(* Schneider Machine Expert - Basic project resolucao, file version 2.7.0.0 *)
(* ProjectInformations: Name=Novo projeto *)

HARDWARE
  Cpu 0: TM221CE24R
  EthernetConfiguration: NetworkName=M221, IpAllocationMode=FixedAddress, IpAddress=0.0.0.0, SubnetMask=0.0.0.0
  SerialLineConfiguration: Baud=Baud19200, Parity=ParityEven, DataBits=DataBits8, StopBits=StopBits1, PhysicalMedium=PhysicalMediumRs485, TransmissionMode=TransmissionModeModbusRtu, SlaveId=1, Addressing=SlaveAddressing
  MastTask: UsePeriodScanMode=false, PeriodScan=100
  FastTask: Period=255
  CpuBehavior: StartingMode=StartAsPreviousState, AutoSaveRamOnEeprom=true, WatchdogPeriod=250

SYMBOLS  (address, symbol, comment, settings)
  %M0       SIG_IN_SEN_A
  %M1       SIG_IN_BOT_A
  %M10      SIG_OUT_EST_A_LIGA
  %M11      SIG_OUT_EST_A_DESL
  %TM0        [Preset=5, Base=OneSecond]
  %I0.0     IN_SEN_A
  %I0.1     IN_BOT_A
  %Q0.1     OUT_EST_A

POU Entradas
  (* SectionNumber=1 *)

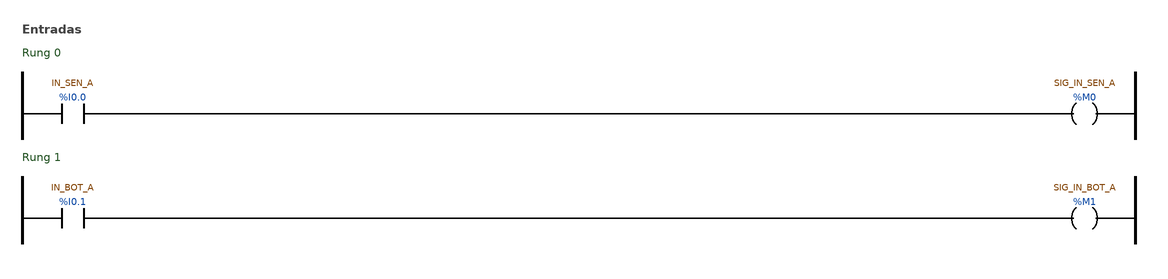

// Rung 0
  LD %I0.0                (* IN_SEN_A *)
  ST %M0                  (* SIG_IN_SEN_A *)
  // as ST:
  //   SIG_IN_SEN_A := IN_SEN_A;

// Rung 1
  LD %I0.1                (* IN_BOT_A *)
  ST %M1                  (* SIG_IN_BOT_A *)
  // as ST:
  //   SIG_IN_BOT_A := IN_BOT_A;

POU Lógicas
  (* SectionNumber=2 *)

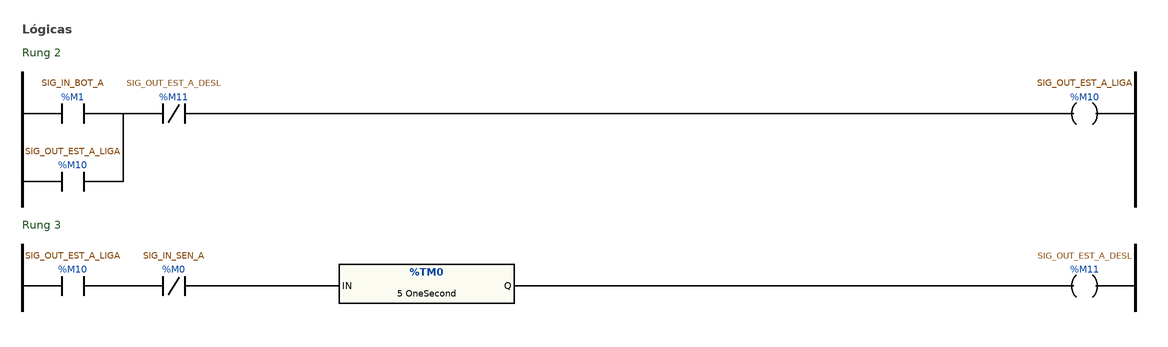

// Rung 2
  LD %M1                  (* SIG_IN_BOT_A *)
  OR %M10                 (* SIG_OUT_EST_A_LIGA *)
  ANDN %M11               (* SIG_OUT_EST_A_DESL *)
  ST %M10                 (* SIG_OUT_EST_A_LIGA *)
  // as ST:
  //   SIG_OUT_EST_A_LIGA := (SIG_IN_BOT_A OR SIG_OUT_EST_A_LIGA) AND NOT SIG_OUT_EST_A_DESL;

// Rung 3
  BLK %TM0
  LD %M10                 (* SIG_OUT_EST_A_LIGA *)
  ANDN %M0                (* SIG_IN_SEN_A *)
  IN
  OUT_BLK
  LD Q
  ST %M11                 (* SIG_OUT_EST_A_DESL *)
  END_BLK
  // as ST:
  //   %TM0(IN := SIG_OUT_EST_A_LIGA AND NOT SIG_IN_SEN_A);
  //   SIG_OUT_EST_A_DESL := %TM0.Q;

POU Saídas
  (* SectionNumber=3 *)

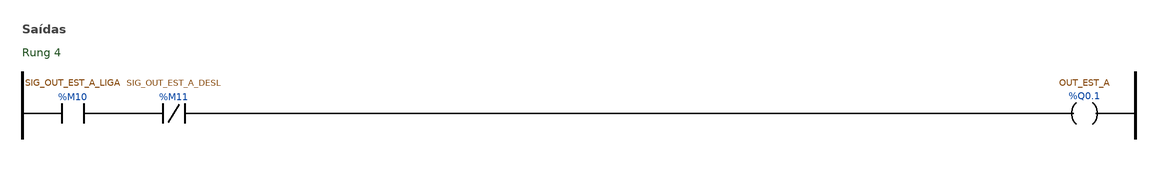

// Rung 4
  LD %M10                 (* SIG_OUT_EST_A_LIGA *)
  ANDN %M11               (* SIG_OUT_EST_A_DESL *)
  ST %Q0.1                (* OUT_EST_A *)
  // as ST:
  //   OUT_EST_A := SIG_OUT_EST_A_LIGA AND NOT SIG_OUT_EST_A_DESL;
